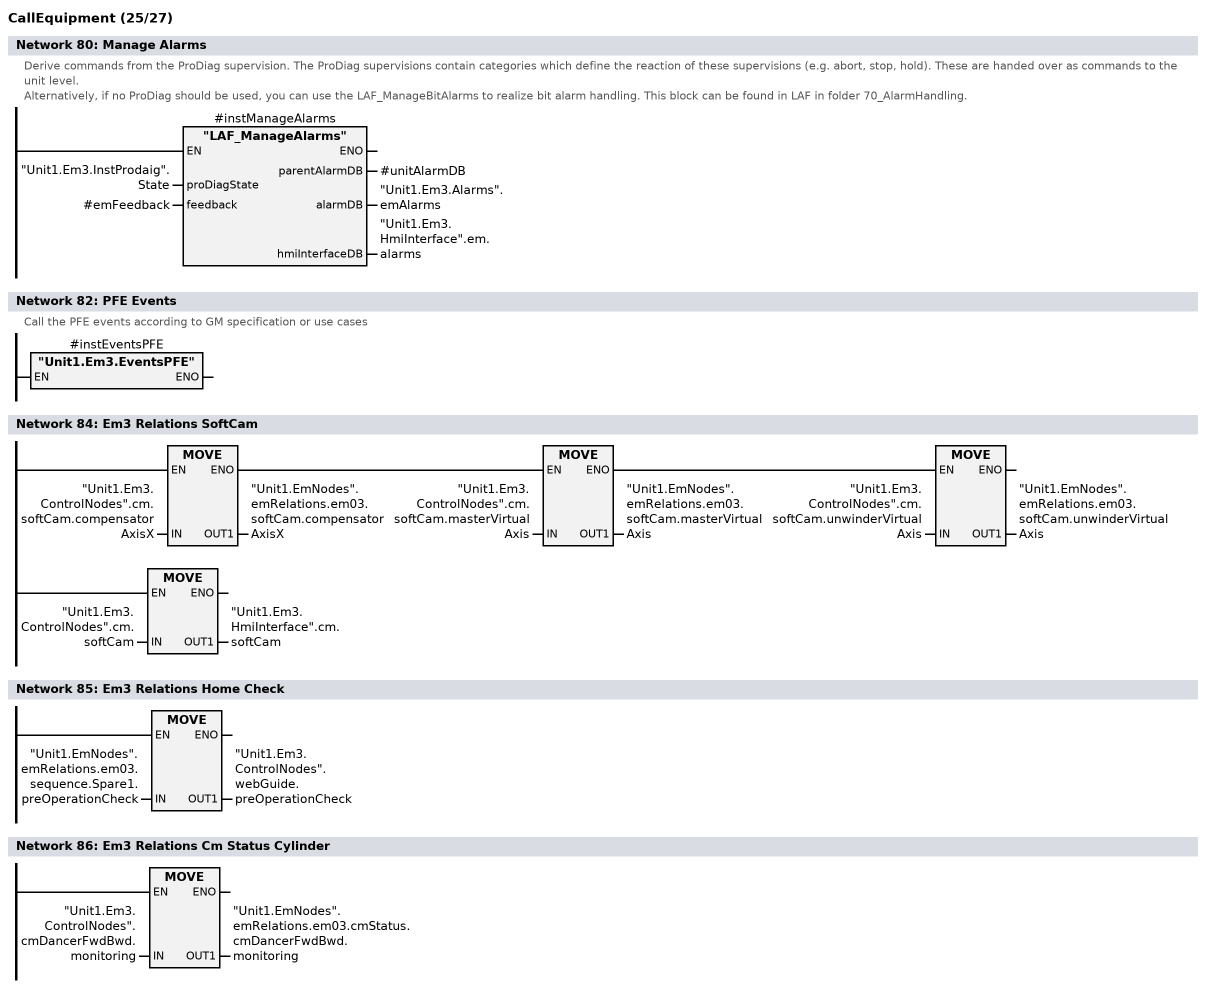
   RUNG wire#powerrail
      #instManageAlarms(proDiagState := "Unit1.Em3.InstProdaig".State, feedback := #emFeedback, parentAlarmDB => #unitAlarmDB, alarmDB => "Unit1.Em3.Alarms".emAlarms, hmiInterfaceDB => "Unit1.Em3.HmiInterface".em.alarms)
   END_RUNG
   // the same network as SCL:
   #instManageAlarms(proDiagState := "Unit1.Em3.InstProdaig".State,   // "LAF_ManageAlarms"
                     feedback := #emFeedback,
                     parentAlarmDB => #unitAlarmDB,
                     alarmDB => "Unit1.Em3.Alarms".emAlarms,
                     hmiInterfaceDB => "Unit1.Em3.HmiInterface".em.alarms);
END_REGION

REGION Network 81: *************** PFE Events**********************************
END_REGION

REGION Network 82: PFE Events
   // Call the PFE events according to GM specification or use cases
   RUNG wire#powerrail
      #instEventsPFE()
   END_RUNG
   // the same network as SCL:
   #instEventsPFE();   // "Unit1.Em3.EventsPFE"
END_REGION

REGION Network 83: ******************** Unit Output ********************
END_REGION

REGION Network 84: Em3 Relations SoftCam
   RUNG wire#powerrail
      Move(in := "Unit1.Em3.ControlNodes".cm.softCam.compensatorAxisX, out1 => "Unit1.EmNodes".emRelations.em03.softCam.compensatorAxisX)
      Move(in := "Unit1.Em3.ControlNodes".cm.softCam.masterVirtualAxis, out1 => "Unit1.EmNodes".emRelations.em03.softCam.masterVirtualAxis)
      Move(in := "Unit1.Em3.ControlNodes".cm.softCam.unwinderVirtualAxis, out1 => "Unit1.EmNodes".emRelations.em03.softCam.unwinderVirtualAxis)
   END_RUNG
   RUNG wire#powerrail
      Move(in := "Unit1.Em3.ControlNodes".cm.softCam, out1 => "Unit1.Em3.HmiInterface".cm.softCam)
   END_RUNG
   // the same network as SCL:
   "Unit1.EmNodes".emRelations.em03.softCam.compensatorAxisX := "Unit1.Em3.ControlNodes".cm.softCam.compensatorAxisX;
   "Unit1.EmNodes".emRelations.em03.softCam.masterVirtualAxis := "Unit1.Em3.ControlNodes".cm.softCam.masterVirtualAxis;
   "Unit1.EmNodes".emRelations.em03.softCam.unwinderVirtualAxis := "Unit1.Em3.ControlNodes".cm.softCam.unwinderVirtualAxis;
   "Unit1.Em3.HmiInterface".cm.softCam := "Unit1.Em3.ControlNodes".cm.softCam;
END_REGION

REGION Network 85: Em3 Relations Home Check
   RUNG wire#powerrail
      Move(in := "Unit1.EmNodes".emRelations.em03.sequence.Spare1.preOperationCheck, out1 => "Unit1.Em3.ControlNodes".webGuide.preOperationCheck)
   END_RUNG
   // the same network as SCL:
   "Unit1.Em3.ControlNodes".webGuide.preOperationCheck := "Unit1.EmNodes".emRelations.em03.sequence.Spare1.preOperationCheck;
END_REGION

REGION Network 86: Em3 Relations Cm Status Cylinder
   RUNG wire#powerrail
      Move(in := "Unit1.Em3.ControlNodes".cmDancerFwdBwd.monitoring, out1 => "Unit1.EmNodes".emRelations.em03.cmStatus.cmDancerFwdBwd.monitoring)
   END_RUNG
   // the same network as SCL:
   "Unit1.EmNodes".emRelations.em03.cmStatus.cmDancerFwdBwd.monitoring := "Unit1.Em3.ControlNodes".cmDancerFwdBwd.monitoring;
END_REGION

REGION Network 87: Em3 Relations CmStatus Digital Signal
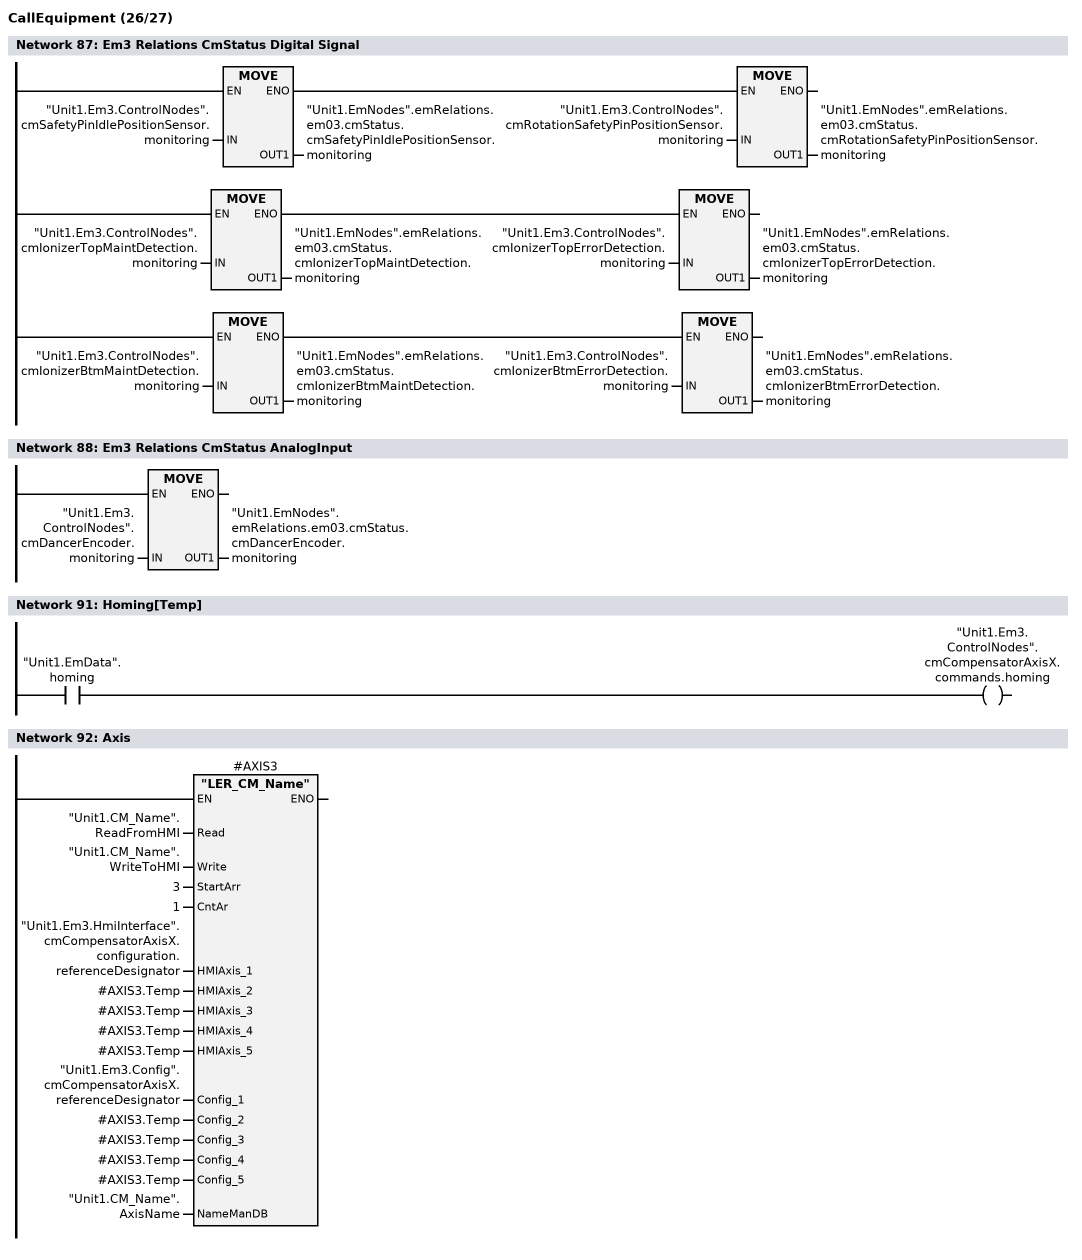
   RUNG wire#powerrail
      Move(in := "Unit1.Em3.ControlNodes".cmSafetyPinIdlePositionSensor.monitoring, out1 => "Unit1.EmNodes".emRelations.em03.cmStatus.cmSafetyPinIdlePositionSensor.monitoring)
      Move(in := "Unit1.Em3.ControlNodes".cmRotationSafetyPinPositionSensor.monitoring, out1 => "Unit1.EmNodes".emRelations.em03.cmStatus.cmRotationSafetyPinPositionSensor.monitoring)
   END_RUNG
   RUNG wire#powerrail
      Move(in := "Unit1.Em3.ControlNodes".cmIonizerTopMaintDetection.monitoring, out1 => "Unit1.EmNodes".emRelations.em03.cmStatus.cmIonizerTopMaintDetection.monitoring)
      Move(in := "Unit1.Em3.ControlNodes".cmIonizerTopErrorDetection.monitoring, out1 => "Unit1.EmNodes".emRelations.em03.cmStatus.cmIonizerTopErrorDetection.monitoring)
   END_RUNG
   RUNG wire#powerrail
      Move(in := "Unit1.Em3.ControlNodes".cmIonizerBtmMaintDetection.monitoring, out1 => "Unit1.EmNodes".emRelations.em03.cmStatus.cmIonizerBtmMaintDetection.monitoring)
      Move(in := "Unit1.Em3.ControlNodes".cmIonizerBtmErrorDetection.monitoring, out1 => "Unit1.EmNodes".emRelations.em03.cmStatus.cmIonizerBtmErrorDetection.monitoring)
   END_RUNG
   // the same network as SCL:
   "Unit1.EmNodes".emRelations.em03.cmStatus.cmSafetyPinIdlePositionSensor.monitoring := "Unit1.Em3.ControlNodes".cmSafetyPinIdlePositionSensor.monitoring;
   "Unit1.EmNodes".emRelations.em03.cmStatus.cmRotationSafetyPinPositionSensor.monitoring := "Unit1.Em3.ControlNodes".cmRotationSafetyPinPositionSensor.monitoring;
   "Unit1.EmNodes".emRelations.em03.cmStatus.cmIonizerTopMaintDetection.monitoring := "Unit1.Em3.ControlNodes".cmIonizerTopMaintDetection.monitoring;
   "Unit1.EmNodes".emRelations.em03.cmStatus.cmIonizerTopErrorDetection.monitoring := "Unit1.Em3.ControlNodes".cmIonizerTopErrorDetection.monitoring;
   "Unit1.EmNodes".emRelations.em03.cmStatus.cmIonizerBtmMaintDetection.monitoring := "Unit1.Em3.ControlNodes".cmIonizerBtmMaintDetection.monitoring;
   "Unit1.EmNodes".emRelations.em03.cmStatus.cmIonizerBtmErrorDetection.monitoring := "Unit1.Em3.ControlNodes".cmIonizerBtmErrorDetection.monitoring;
END_REGION

REGION Network 88: Em3 Relations CmStatus AnalogInput
   RUNG wire#powerrail
      Move(in := "Unit1.Em3.ControlNodes".cmDancerEncoder.monitoring, out1 => "Unit1.EmNodes".emRelations.em03.cmStatus.cmDancerEncoder.monitoring)
   END_RUNG
   // the same network as SCL:
   "Unit1.EmNodes".emRelations.em03.cmStatus.cmDancerEncoder.monitoring := "Unit1.Em3.ControlNodes".cmDancerEncoder.monitoring;
END_REGION

REGION Network 89: Em3 Relations Select Job Status
END_REGION

REGION Network 90: Em3 Relations Sequence Interface
END_REGION

REGION Network 91: Homing[Temp]
   RUNG wire#powerrail
      Contact( "Unit1.EmData".homing )
      Coil( "Unit1.Em3.ControlNodes".cmCompensatorAxisX.commands.homing )
   END_RUNG
   // the same network as SCL:
   "Unit1.Em3.ControlNodes".cmCompensatorAxisX.commands.homing := "Unit1.EmData".homing;
END_REGION

REGION Network 92: Axis
   RUNG wire#powerrail
      #AXIS3(Read := "Unit1.CM_Name".ReadFromHMI, Write := "Unit1.CM_Name".WriteToHMI, StartArr := 3, CntAr := 1, HMIAxis_1 := "Unit1.Em3.HmiInterface".cmCompensatorAxisX.configuration.referenceDesignator, HMIAxis_2 := #AXIS3.Temp, HMIAxis_3 := #AXIS3.Temp, HMIAxis_4 := #AXIS3.Temp, HMIAxis_5 := #AXIS3.Temp, Config_1 := "Unit1.Em3.Config".cmCompensatorAxisX.referenceDesignator, Config_2 := #AXIS3.Temp, Config_3 := #AXIS3.Temp, Config_4 := #AXIS3.Temp, Config_5 := #AXIS3.Temp, NameManDB := "Unit1.CM_Name".AxisName)
   END_RUNG
   // the same network as SCL:
   #AXIS3(Read := "Unit1.CM_Name".ReadFromHMI,   // "LER_CM_Name"
          Write := "Unit1.CM_Name".WriteToHMI,
          StartArr := 3,
          CntAr := 1,
          HMIAxis_1 := "Unit1.Em3.HmiInterface".cmCompensatorAxisX.configuration.referenceDesignator,
          HMIAxis_2 := #AXIS3.Temp,
          HMIAxis_3 := #AXIS3.Temp,
          HMIAxis_4 := #AXIS3.Temp,
          HMIAxis_5 := #AXIS3.Temp,
          Config_1 := "Unit1.Em3.Config".cmCompensatorAxisX.referenceDesignator,
          Config_2 := #AXIS3.Temp,
          Config_3 := #AXIS3.Temp,
          Config_4 := #AXIS3.Temp,
          Config_5 := #AXIS3.Temp,
          NameManDB := "Unit1.CM_Name".AxisName);
END_REGION

REGION Network 93: Cylinder
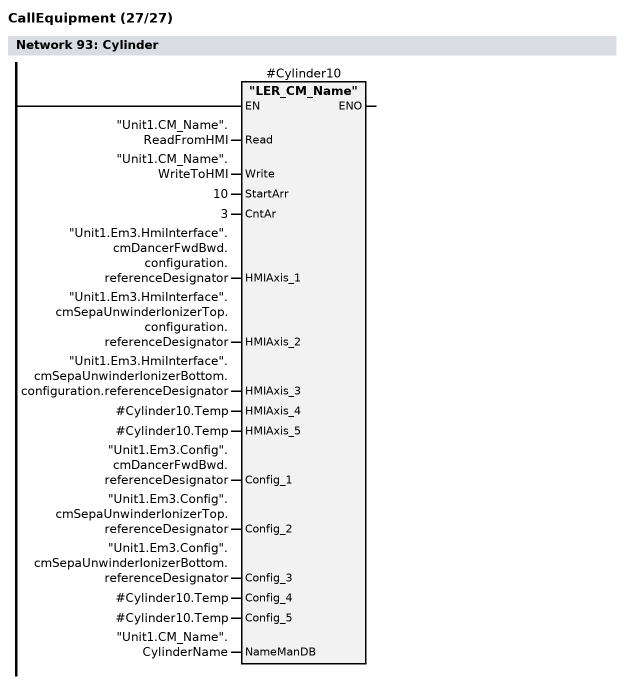
   RUNG wire#powerrail
      #Cylinder10(Read := "Unit1.CM_Name".ReadFromHMI, Write := "Unit1.CM_Name".WriteToHMI, StartArr := 10, CntAr := 3, HMIAxis_1 := "Unit1.Em3.HmiInterface".cmDancerFwdBwd.configuration.referenceDesignator, HMIAxis_2 := "Unit1.Em3.HmiInterface".cmSepaUnwinderIonizerTop.configuration.referenceDesignator, HMIAxis_3 := "Unit1.Em3.HmiInterface".cmSepaUnwinderIonizerBottom.configuration.referenceDesignator, HMIAxis_4 := #Cylinder10.Temp, HMIAxis_5 := #Cylinder10.Temp, Config_1 := "Unit1.Em3.Config".cmDancerFwdBwd.referenceDesignator, Config_2 := "Unit1.Em3.Config".cmSepaUnwinderIonizerTop.referenceDesignator, Config_3 := "Unit1.Em3.Config".cmSepaUnwinderIonizerBottom.referenceDesignator, Config_4 := #Cylinder10.Temp, Config_5 := #Cylinder10.Temp, NameManDB := "Unit1.CM_Name".CylinderName)
   END_RUNG
   // the same network as SCL:
   #Cylinder10(Read := "Unit1.CM_Name".ReadFromHMI,   // "LER_CM_Name"
               Write := "Unit1.CM_Name".WriteToHMI,
               StartArr := 10,
               CntAr := 3,
               HMIAxis_1 := "Unit1.Em3.HmiInterface".cmDancerFwdBwd.configuration.referenceDesignator,
               HMIAxis_2 := "Unit1.Em3.HmiInterface".cmSepaUnwinderIonizerTop.configuration.referenceDesignator,
               HMIAxis_3 := "Unit1.Em3.HmiInterface".cmSepaUnwinderIonizerBottom.configuration.referenceDesignator,
               HMIAxis_4 := #Cylinder10.Temp,
               HMIAxis_5 := #Cylinder10.Temp,
               Config_1 := "Unit1.Em3.Config".cmDancerFwdBwd.referenceDesignator,
               Config_2 := "Unit1.Em3.Config".cmSepaUnwinderIonizerTop.referenceDesignator,
               Config_3 := "Unit1.Em3.Config".cmSepaUnwinderIonizerBottom.referenceDesignator,
               Config_4 := #Cylinder10.Temp,
               Config_5 := #Cylinder10.Temp,
               NameManDB := "Unit1.CM_Name".CylinderName);
END_REGION
END_FUNCTION_BLOCK
